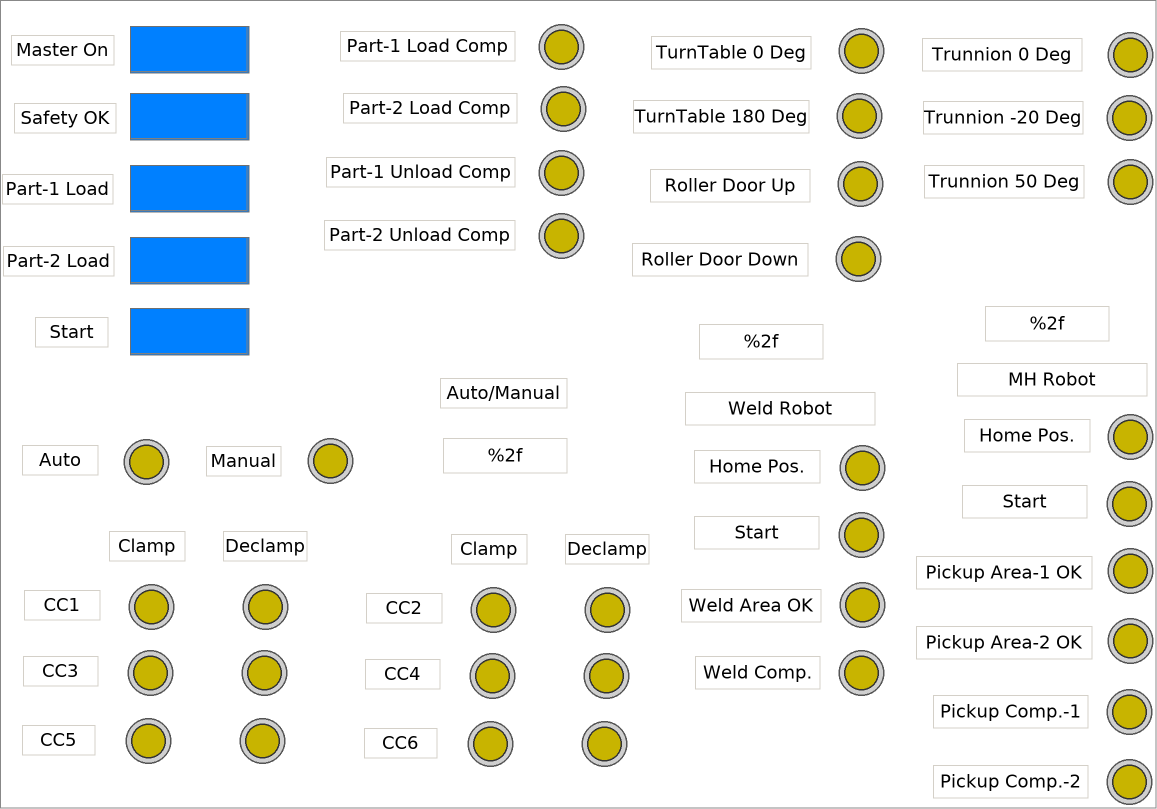
VISUALIZATION Auto_Cycle_Fix2  // 1157x809
    Textfield (340,31 175x30), "Part-1 Load Comp"
    Textfield (343,93 174x30), "Part-2 Load Comp"
    Lamp1 (537,82 53x54), variable: Auto_Cycle_Fix2.Fixture_2.Part2_Load_Comp, style: Lamp-Lamp1-Yellow
    Textfield (651,36 160x33), "TurnTable 0 Deg"
    Lamp1 (835,24 53x54), variable: Auto_Cycle_Fix2.TurnTable_1.TT_0_Deg, style: Lamp-Lamp1-Yellow
    Textfield (633,100 176x33), "TurnTable 180 Deg"
    Lamp1 (833,89 53x54), variable: Auto_Cycle_Fix2.TurnTable_1.TT_180_Deg, style: Lamp-Lamp1-Yellow
    Textfield (922,38 160x33), "Trunnion 0 Deg"
    Lamp1 (1104,28 53x54), variable: Auto_Cycle_Fix2.Trunnion_1.TR_0_Deg, style: Lamp-Lamp1-Yellow
    Textfield (923,101 160x33), "Trunnion -20 Deg"
    Lamp1 (1103,91 53x54), variable: Auto_Cycle_Fix2.Trunnion_1.TR_20_Deg, style: Lamp-Lamp1-Yellow
    Lamp1 (1104,155 53x54), variable: Auto_Cycle_Fix2.Trunnion_1.TR_50_Deg, style: Lamp-Lamp1-Yellow
    Textfield (924,165 160x33), "Trunnion 50 Deg"
    Textfield (24,590 76x30), "CC1"
    Textfield (23,656 75x30), "CC3"
    Textfield (22,725 73x30), "CC5"
    Lamp1 (125,580 53x54), variable: Auto_Cycle_Fix2.Fixture_2.CC1_Output.Work_Position, style: Lamp-Lamp1-Yellow
    Lamp1 (124,646 53x54), variable: Auto_Cycle_Fix2.Fixture_2.CC3_Output.Work_Position, style: Lamp-Lamp1-Yellow
    Lamp1 (122,714 53x54), variable: Auto_Cycle_Fix2.Fixture_2.CC5_Output.Work_Position, style: Lamp-Lamp1-Yellow
    Textfield (109,531 76x30), "Clamp"
    Lamp1 (239,580 53x54), variable: Auto_Cycle_Fix2.Fixture_2.CC1_Output.Home_Position, style: Lamp-Lamp1-Yellow
    Lamp1 (238,646 53x54), variable: Auto_Cycle_Fix2.Fixture_2.CC3_Output.Home_Position, style: Lamp-Lamp1-Yellow
    Lamp1 (236,714 53x54), variable: Auto_Cycle_Fix2.Fixture_2.CC5_Output.Home_Position, style: Lamp-Lamp1-Yellow
    Textfield (223,531 84x30), "Declamp"
    Textfield (366,593 76x30), "CC2"
    Textfield (365,659 75x30), "CC4"
    Textfield (364,728 73x30), "CC6"
    Lamp1 (467,583 53x54), variable: Auto_Cycle_Fix2.Fixture_2.CC2_Output.Work_Position, style: Lamp-Lamp1-Yellow
    Lamp1 (466,649 53x54), variable: Auto_Cycle_Fix2.Fixture_2.CC4_Output.Work_Position, style: Lamp-Lamp1-Yellow
    Lamp1 (464,717 53x54), variable: Auto_Cycle_Fix2.Fixture_2.CC6_Output.Work_Position, style: Lamp-Lamp1-Yellow
    Textfield (451,534 76x30), "Clamp"
    Lamp1 (581,583 53x54), variable: Auto_Cycle_Fix2.Fixture_2.CC2_Output.Home_Position, style: Lamp-Lamp1-Yellow
    Lamp1 (580,649 53x54), variable: Auto_Cycle_Fix2.Fixture_2.CC4_Output.Home_Position, style: Lamp-Lamp1-Yellow
    Lamp1 (578,717 53x54), variable: Auto_Cycle_Fix2.Fixture_2.CC6_Output.Home_Position, style: Lamp-Lamp1-Yellow
    Textfield (565,534 84x30), "Declamp"
    Textfield (22,445 76x30), "Auto"
    Textfield (206,446 75x30), "Manual"
    Lamp1 (304,434 53x54), variable: Manual_Mode, style: Lamp-Lamp1-Yellow
    Textfield (650,169 160x33), "Roller Door Up"
    Lamp1 (834,157 53x54), variable: Auto_Cycle_Fix2.RollerDoor_1.Roller_Up, style: Lamp-Lamp1-Yellow
    Textfield (632,243 176x33), "Roller Door Down"
    Lamp1 (832,232 53x54), variable: Auto_Cycle_Fix2.RollerDoor_1.Roller_Down, style: Lamp-Lamp1-Yellow
    Textfield (694,450 126x33), "Home Pos."
    Lamp1 (836,441 53x54), variable: Auto_Cycle_Fix2.Robot_Weld_1.Robot_1_In.i_Home, style: Lamp-Lamp1-Yellow
    Textfield (681,589 140x33), "Weld Area OK"
    Lamp1 (836,578 53x54), variable: Auto_Cycle_Fix2.Robot_Weld_1.Robot_1_In.i_Area_Ok, style: Lamp-Lamp1-Yellow
    Textfield (695,656 125x33), "Weld Comp."
    Lamp1 (835,646 53x54), variable: Auto_Cycle_Fix2.Robot_Weld_1.Robot_1_Out.o_Weld_Comp, style: Lamp-Lamp1-Yellow
    Textfield (685,392 190x33), "Weld Robot"
    Textfield (957,363 190x33), "MH Robot"
    Textfield (694,516 125x33), "Start"
    Lamp1 (835,508 53x54), variable: Auto_Cycle_Fix2.Robot_Weld_1.Robot_1_In.i_Start, style: Lamp-Lamp1-Yellow
    Textfield (964,419 126x33), "Home Pos."
    Lamp1 (1104,410 53x54), variable: Auto_Cycle_Fix2.Robot_MH_1.Robot_1_In.i_Home, style: Lamp-Lamp1-Yellow
    Textfield (916,556 176x33), "Pickup Area-1 OK"
    Lamp1 (1104,544 53x54), variable: Auto_Cycle_Fix2.Robot_MH_1.Robot_1_In.i_Area_Ok1, style: Lamp-Lamp1-Yellow
    Textfield (933,695 155x33), "Pickup Comp.-1"
    Lamp1 (1103,685 53x54), variable: Auto_Cycle_Fix2.Robot_MH_1.Robot_1_Out.o_Pickup_Comp1, style: Lamp-Lamp1-Yellow
    Textfield (962,485 125x33), "Start"
    Lamp1 (1103,477 53x54), variable: Auto_Cycle_Fix2.Robot_MH_1.Robot_1_In.i_Start, style: Lamp-Lamp1-Yellow
    Textfield (2,174 111x30), "Part-1 Load"
    Button (130,165 119x47)
        p573394764: Fix2_Part_1_Load
        toggle Fix2_Part_1_Load
    Textfield (440,378 127x30), "Auto/Manual"
    Textfield (326,157 189x30), "Part-1 Unload Comp"
    Lamp1 (535,146 53x54), variable: Auto_Cycle_Fix2.Fixture_2.Part1_Unload_Comp, style: Lamp-Lamp1-Yellow
    Textfield (324,220 191x30), "Part-2 Unload Comp"
    Lamp1 (535,209 53x54), variable: Auto_Cycle_Fix2.Fixture_2.Part2_Unload_Comp, style: Lamp-Lamp1-Yellow
    Textfield (443,438 124x35), "%2f", text variable: Station_Mode
        OnMouseDown: write Station_Mode via VisuDialogs.Numpad
    Textfield (916,626 176x33), "Pickup Area-2 OK"
    Lamp1 (1104,614 53x54), variable: Auto_Cycle_Fix2.Robot_MH_1.Robot_1_In.i_Area_Ok2, style: Lamp-Lamp1-Yellow
    Textfield (933,765 155x33), "Pickup Comp.-2"
    Lamp1 (1103,755 53x54), variable: Auto_Cycle_Fix2.Robot_MH_1.Robot_1_Out.o_Pickup_Comp2, style: Lamp-Lamp1-Yellow
    Lamp1 (120,435 53x54), variable: Auto_Mode, style: Lamp-Lamp1-Yellow
    Textfield (11,35 103x30), "Master On"
    Button (130,26 119x47)
        p573394764: Master_On
        toggle Master_On
    Textfield (14,103 102x30), "Safety OK"
    Button (130,93 119x47)
        p573394764: Safety_Ok
        toggle Safety_Ok
    Textfield (3,246 111x30), "Part-2 Load"
    Button (130,237 119x47)
        p573394764: Fix2_Part_2_Load
        toggle Fix2_Part_2_Load
    Textfield (35,317 73x30), "Start"
    Button (130,308 119x47)
        p573394764: Start_Pb
        tap Start_Pb
    Textfield (699,324 124x35), "%2f", text variable: Auto_Cycle_Fix2.Robot_Weld_1.Robot_1_In.i_Prg_No
        OnMouseDown: write Auto_Cycle_Fix2.Robot_Weld_1.Robot_1_In.i_Prg_No via VisuDialogs.Numpad
    Textfield (985,306 124x35), "%2f", text variable: Auto_Cycle_Fix2.Robot_MH_1.Robot_1_In.i_Prg_No
        OnMouseDown: write Auto_Cycle_Fix2.Robot_MH_1.Robot_1_In.i_Prg_No via VisuDialogs.Numpad
    Lamp1 (535,20 53x54), variable: Auto_Cycle_Fix2.Fixture_2.Part1_Load_Comp, style: Lamp-Lamp1-Yellow
END_VISUALIZATION

(* stored: Version 1.1.0.1, ProductVersion 3.1.4024.16
   Visu Auto_Cycle_Fix2: Id {73535c92-cec9-4923-a398-3e8ad8034d0e} *)
